TYPE ST_DigitalInput :
STRUCT
	hmi_In: BOOL;
	i_In AT %I* : BOOL;
	mode: E_Mode;
END_STRUCT
END_TYPE

(* stored: Version 1.1.0.1, ProductVersion 3.1.4024.12
   DUT ST_DigitalInput: Id {b43f835c-b5a2-4009-8649-f277eb23ef52} *)
